ABB RobotStudio station: Sjenk-o-bot.rsstn

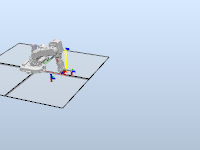
Station Lab3 (saved by RobotStudio 21.2.9526.0)
Controller IRB140_6_81
  mechanical unit ROB_1: IRB140_6_81_C_03, 6 joints, base frame (0, 0, 0) mm
Layout (positions relative to the parent item):
  - IRB140_6_81_C_03 [mechanism, from Robots\IRB140_6_81_C_G_03.rslib] at (0, 0, 0) mm; joint values [0, 1.2298, 0.1403, 3.1416, 1.3702, 2.3736] (rad or m)
  - Griper [mechanism] at (550, 0, 100) mm, rotated rx -90 ry 46 rz -90 deg; joint values [0, 0] (rad or m)
      TCP Griper_1 at (0, 0, 130) mm, rotated rx 0 ry 0 rz -90 deg
      links: L1, L2, L3
Attachment: Griper is attached to IRB140_6_81_C_03 / Link6
EventTableEntry 1023: Group=, Trigger=DO10_2 1024, Actions=[EventTableActionMechanicalPose 1025], Comment=, ActivationMode=2, Cyclic=false
EventTableTriggerIO 1024: IOValue=[1], IRC5Controller=? -1, Operator=0, SignalSource=IRB140_6_81 515
EventTableActionMechanicalPose 1025: VirtualSignal=, Mechanism=Griper 1017, ToPoseName=EndPose, VirtualSignalValue=[1]
EventTableEntry 1026: Group=, Trigger=DO10_2 1027, Actions=[EventTableActionMechanicalPose 1028], Comment=, ActivationMode=2, Cyclic=false
EventTableTriggerIO 1027: IOValue=[0], IRC5Controller=? -1, Operator=0, SignalSource=IRB140_6_81 515
EventTableActionMechanicalPose 1028: VirtualSignal=, Mechanism=Griper 1017, ToPoseName=HomePosition, VirtualSignalValue=[1]
EventTableTriggerIO 1037: IOValue=[1], IRC5Controller=? -1, Operator=0, SignalSource=IRB140_6_81 515
EventTableTriggerIO 1038: IOValue=[0], IRC5Controller=? -1, Operator=0, SignalSource=IRB140_6_81 515
EventTableTriggerIO 1074: IOValue=[1], IRC5Controller=? -1, Operator=0, SignalSource=IRB140_6_81 515
EventTableTriggerIO 1075: IOValue=[1], IRC5Controller=? -1, Operator=0, SignalSource=IRB140_6_81 515
EventTableTriggerIO 1076: IOValue=[1], IRC5Controller=? -1, Operator=0, SignalSource=IRB140_6_81 515
EventTableTriggerIO 1077: IOValue=[1], IRC5Controller=? -1, Operator=0, SignalSource=IRB140_6_81 515
EventTableTriggerIO 1078: IOValue=[1], IRC5Controller=? -1, Operator=0, SignalSource=IRB140_6_81 515
EventTableTriggerIO 1079: IOValue=[0], IRC5Controller=? -1, Operator=0, SignalSource=IRB140_6_81 515
EventTableTriggerIO 1080: IOValue=[0], IRC5Controller=? -1, Operator=0, SignalSource=IRB140_6_81 515
EventTableTriggerIO 1081: IOValue=[0], IRC5Controller=? -1, Operator=0, SignalSource=IRB140_6_81 515
EventTableTriggerIO 1082: IOValue=[0], IRC5Controller=? -1, Operator=0, SignalSource=IRB140_6_81 515
EventTableTriggerIO 1083: IOValue=[0], IRC5Controller=? -1, Operator=0, SignalSource=IRB140_6_81 515
EventTableTriggerIO 1113: IOValue=[1], IRC5Controller=? -1, Operator=0, SignalSource=IRB140_6_81 515
EventTableTriggerIO 1114: IOValue=[0], IRC5Controller=? -1, Operator=0, SignalSource=IRB140_6_81 515
EventTableTriggerIO 1152: IOValue=[1], IRC5Controller=? -1, Operator=0, SignalSource=IRB140_6_81 515
EventTableTriggerIO 1153: IOValue=[0], IRC5Controller=? -1, Operator=0, SignalSource=IRB140_6_81 515
EventTableTriggerIO 1154: IOValue=[1], IRC5Controller=? -1, Operator=0, SignalSource=IRB140_6_81 515
EventTableTriggerIO 1155: IOValue=[1], IRC5Controller=? -1, Operator=0, SignalSource=IRB140_6_81 515
EventTableTriggerIO 1156: IOValue=[1], IRC5Controller=? -1, Operator=0, SignalSource=IRB140_6_81 515
EventTableTriggerIO 1157: IOValue=[1], IRC5Controller=? -1, Operator=0, SignalSource=IRB140_6_81 515
EventTableTriggerIO 1158: IOValue=[0], IRC5Controller=? -1, Operator=0, SignalSource=IRB140_6_81 515
EventTableTriggerIO 1159: IOValue=[0], IRC5Controller=? -1, Operator=0, SignalSource=IRB140_6_81 515
EventTableTriggerIO 1160: IOValue=[0], IRC5Controller=? -1, Operator=0, SignalSource=IRB140_6_81 515
EventTableTriggerIO 1161: IOValue=[0], IRC5Controller=? -1, Operator=0, SignalSource=IRB140_6_81 515
EventTableTriggerIO 1197: IOValue=[1], IRC5Controller=? -1, Operator=0, SignalSource=IRB140_6_81 515
EventTableTriggerIO 1198: IOValue=[1], IRC5Controller=? -1, Operator=0, SignalSource=IRB140_6_81 515
EventTableTriggerIO 1199: IOValue=[1], IRC5Controller=? -1, Operator=0, SignalSource=IRB140_6_81 515
EventTableTriggerIO 1200: IOValue=[1], IRC5Controller=? -1, Operator=0, SignalSource=IRB140_6_81 515
EventTableTriggerIO 1201: IOValue=[1], IRC5Controller=? -1, Operator=0, SignalSource=IRB140_6_81 515
EventTableTriggerIO 1202: IOValue=[0], IRC5Controller=? -1, Operator=0, SignalSource=IRB140_6_81 515
EventTableTriggerIO 1203: IOValue=[0], IRC5Controller=? -1, Operator=0, SignalSource=IRB140_6_81 515
EventTableTriggerIO 1204: IOValue=[0], IRC5Controller=? -1, Operator=0, SignalSource=IRB140_6_81 515
EventTableTriggerIO 1205: IOValue=[0], IRC5Controller=? -1, Operator=0, SignalSource=IRB140_6_81 515
EventTableTriggerIO 1206: IOValue=[0], IRC5Controller=? -1, Operator=0, SignalSource=IRB140_6_81 515
EventTableTriggerIO 1240: IOValue=[1], IRC5Controller=? -1, Operator=0, SignalSource=IRB140_6_81 515
EventTableTriggerIO 1241: IOValue=[0], IRC5Controller=? -1, Operator=0, SignalSource=IRB140_6_81 515
EventTableTriggerIO 1297: IOValue=[1], IRC5Controller=? -1, Operator=0, SignalSource=IRB140_6_81 515
EventTableTriggerIO 1298: IOValue=[1], IRC5Controller=? -1, Operator=0, SignalSource=IRB140_6_81 515
EventTableTriggerIO 1299: IOValue=[1], IRC5Controller=? -1, Operator=0, SignalSource=IRB140_6_81 515
EventTableTriggerIO 1300: IOValue=[0], IRC5Controller=? -1, Operator=0, SignalSource=IRB140_6_81 515
EventTableTriggerIO 1301: IOValue=[0], IRC5Controller=? -1, Operator=0, SignalSource=IRB140_6_81 515
EventTableTriggerIO 1302: IOValue=[0], IRC5Controller=? -1, Operator=0, SignalSource=IRB140_6_81 515
EventTableTriggerIO 1303: IOValue=[1], IRC5Controller=? -1, Operator=0, SignalSource=IRB140_6_81 515
EventTableTriggerIO 1304: IOValue=[1], IRC5Controller=? -1, Operator=0, SignalSource=IRB140_6_81 515
EventTableTriggerIO 1305: IOValue=[0], IRC5Controller=? -1, Operator=0, SignalSource=IRB140_6_81 515
EventTableTriggerIO 1306: IOValue=[0], IRC5Controller=? -1, Operator=0, SignalSource=IRB140_6_81 515
EventTableTriggerIO 1307: IOValue=[1], IRC5Controller=? -1, Operator=0, SignalSource=IRB140_6_81 515
EventTableTriggerIO 1308: IOValue=[0], IRC5Controller=? -1, Operator=0, SignalSource=IRB140_6_81 515
EventTableTriggerIO 2007: IOValue=[1], IRC5Controller=? -1, Operator=0, SignalSource=IRB140_6_81 515
EventTableTriggerIO 2008: IOValue=[0], IRC5Controller=? -1, Operator=0, SignalSource=IRB140_6_81 515
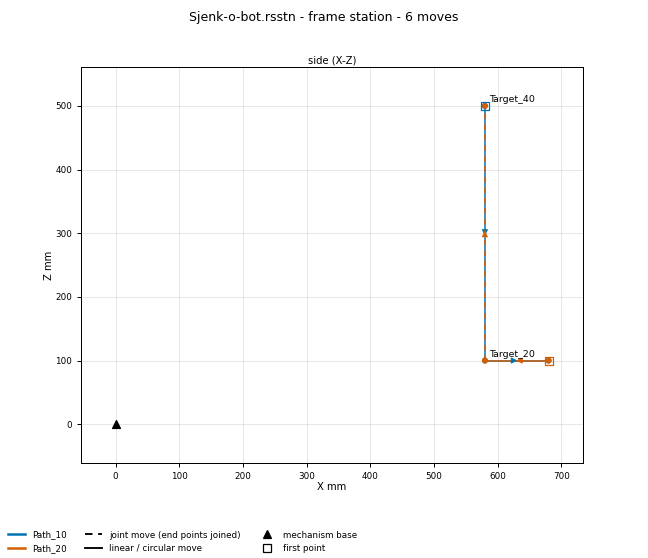
[picture p0: tool path of Sjenk-o-bot.rsstn in frame station, 6 of 22 moves have a stored position in this frame; points joined in program order, loops and branches not executed]
Targets, tools, work objects and paths stored in the station, written as RAPID:
! task T_ROB1
MODULE CalibData
  PERS tooldata Griper_1:=[TRUE,[[0,0,130],[0.927183855,0,0,0.374606593]],[1,[1,1,1],[1,0,0,0],0,0,0]];
  TASK PERS wobjdata Workobject_3:=[FALSE,TRUE,"",[[0,0,0],[1,0,0,0]],[[480,-360,100],[0.707106781,0,0.707106781,0]]];
  PERS wobjdata Workobject_1:=[FALSE,TRUE,"",[[500,0,0],[1,0,0,0]],[[0,0,0],[1,0,0,0]]];
  TASK PERS wobjdata Workobject_2:=[FALSE,TRUE,"",[[0,0,0],[1,0,0,0]],[[480,-360,100],[1,0,0,0]]];
ENDMODULE

! task T_ROB1
MODULE Module1
  CONST robtarget Target_10:=[[0,0,0],[1,0,0,0],[0,0,0,0],[9E+09,9E+09,9E+09,9E+09,9E+09,9E+09]];
  CONST robtarget Target_20:=[[0,360,100],[1,0,0,0],[0,2,2,0],[9E+09,9E+09,9E+09,9E+09,9E+09,9E+09]];
  CONST robtarget Target_30:=[[0,360,200],[1,0,0,0],[0,2,2,0],[9E+09,9E+09,9E+09,9E+09,9E+09,9E+09]];
  CONST robtarget Target_40:=[[-400,360,100],[1,0,0,0],[0,2,2,0],[9E+09,9E+09,9E+09,9E+09,9E+09,9E+09]];
  PROC Path_10()
    MoveJ Target_40,v100,z100,Griper_1\WObj:=Workobject_3;
    WaitTime 2;
    Set DO10_3;
    Reset DO10_2;
    WaitTime 2;
    MoveL Target_20,v100,z100,Griper_1\WObj:=Workobject_3;
    WaitTime 2;
    MoveL Target_30,v100,z100,Griper_1\WObj:=Workobject_3;
    WaitTime 2;
    Set DO10_2;
    Reset DO10_3;
    WaitTime 2;
  ENDPROC
  PROC Path_20()
    MoveL Target_30,v100,z100,Griper_1\WObj:=Workobject_3;
    WaitTime 2;
    Set DO10_3;
    Reset DO10_2;
    WaitTime 2;
    MoveL Target_20,v100,z100,Griper_1\WObj:=Workobject_3;
    WaitTime 2;
    MoveJ Target_40,v100,z100,Griper_1\WObj:=Workobject_3;
  ENDPROC
ENDMODULE

! task T_ROB1
MODULE MainModule
  VAR robtarget home:=[[0,0,0],[1,0,0,0],[0,0,0,0],[9E+09,9E+09,9E+09,9E+09,9E+09,9E+09]];
  PROC main()
    Path_10;
    MoveL RelTool(delivery, -200, 120*0.707106781-32, -120*0.707106781-20 \Rx:=-45),v100,z100,Griper_1\WObj:=Workobject_3;
    MoveL RelTool(delivery, 0, 120*0.707106781-32, -120*0.707106781-20 \Rx:=-45),v100,z100,Griper_1\WObj:=Workobject_3;
    WaitTime 2;
    MoveJ RelTool(delivery, 0, 120*0.707106781-32, -120*0.707106781-20 \Rx:=-45 \Rz:=105),v20\T:=3,fine,Griper_1\WObj:=Workobject_3;
    WaitTime 3;
    MoveJ RelTool(delivery, 0, 120*0.707106781-32, -120*0.707106781-20 \Rx:=-45 \Rz:=0),v20\T:=3,fine,Griper_1\WObj:=Workobject_3;
    WaitTime 1;
    MoveL RelTool(delivery, -200, 120*0.707106781-32, -120*0.707106781-20 \Rx:=-45),v100,z100,Griper_1\WObj:=Workobject_3;
    MoveL RelTool(delivery, 0, -120*0.707106781-52, 120*0.707106781-10 \Rx:=-45),v100,z100,Griper_1\WObj:=Workobject_3;
    WaitTime 2;
    MoveJ RelTool(delivery, 0, -120*0.707106781-52, 120*0.707106781-10 \Rx:=-45 \Rz:=-105),v20\T:=3,fine,Griper_1\WObj:=Workobject_3;
    WaitTime 3;
    MoveJ RelTool(delivery, 0, -120*0.707106781-52, 120*0.707106781-10 \Rx:=-45 \Rz:=0),v20\T:=3,fine,Griper_1\WObj:=Workobject_3;
    WaitTime 1;
    MoveL RelTool(delivery, -200, 120*0.707106781-20, -120*0.707106781-20),v100,z100,Griper_1\WObj:=Workobject_3;
    MoveL RelTool(delivery, 0, 120*0.707106781-20, -120*0.707106781-20),v100,z100,Griper_1\WObj:=Workobject_3;
    WaitTime 2;
    MoveJ RelTool(delivery, 0, 120*0.707106781-20, -120*0.707106781-20 \Rz:=105),v20\T:=3,fine,Griper_1\WObj:=Workobject_3;
    WaitTime 3;
    MoveJ RelTool(delivery, 0, 120*0.707106781-20, -120*0.707106781-20 \Rz:=0),v20\T:=3,fine,Griper_1\WObj:=Workobject_3;
    WaitTime 1;
    MoveL RelTool(delivery, -200, 120*0.707106781-20, -120*0.707106781-20),v100,z100,Griper_1\WObj:=Workobject_3;
    MoveL Offs(delivery, 0, 140, -35),v100,z100,Griper_1\WObj:=Workobject_3;
    WaitTime 2;
    MoveJ RelTool(delivery, 0, 140, -35 \Rz:=105),v20\T:=3,fine,Griper_1\WObj:=Workobject_3;
    WaitTime 3;
    MoveJ RelTool(delivery, 0, 140, -35 \Rz:=0),v20\T:=3,fine,Griper_1\WObj:=Workobject_3;
    WaitTime 1;
    Path_20;
  ENDPROC
ENDMODULE

